// TIA Portal V18 export
TYPE "UDT_AHUsFreshAirCoef"
// stored: IsFailsafeCompliant false
   STRUCT
      IAQ : Array[1..3] of Real;
      Temperature : Array[1..3] of Real;
      BuildingdP : Array[1..3] of Real;
   END_STRUCT;
   // Temperature[1..3] := 1.0;
END_TYPE
